FUNCTION_BLOCK FB_NanotecPD_Power
VAR_INPUT
	bExecute : BOOL;
END_VAR
VAR_OUTPUT
	bBusy 		: BOOL;
	bError 		: BOOL;
	nErrorId 	: ERRORID;	
END_VAR
VAR_IN_OUT
	pHwRef : POINTER TO FB_HwRefNanotecPD; 
END_VAR
VAR
	nState : USINT;
	fbSdoWrite : FB_SDO_WRITE;
END_VAR

//Achtung, anders als bei TMCM-Controllern wird die Statemachine des Controller hier nur bis "SwitchedOn" durchlaufen.
//"OperationEnabled" wird erst nach dem Setzen des Modes gesetzt. Jedes Ändern des Modes erfordert eine Rückkehr zu "SwitchedOn"
IF bExecute THEN
	IF nState = 0 THEN
		bBusy := TRUE;
		CASE pHwRef^.M_GetDS402State() OF
			E_CoDS402States.DS402STATE_Fault:
				pHwRef^.nControlword := 153;	//Reset Error
			E_CoDS402States.DS402STATE_SwitchOnDisabled:
				nState := 1;
			E_CoDS402States.DS402STATE_ReadyToSwitchOn:
				pHwRef^.nControlword := 0;	//Transition 7 in DS402 statemachine -> geht in Switch on disabled
				nState := 1;
			E_CoDS402States.DS402STATE_SwitchedOn:
				pHwRef^.nControlword := 0;	//Transition 10 in DS402 statemachine -> geht in Switch on disabled
				nState := 1;
			E_CoDS402States.DS402STATE_OperationEnabled:
				pHwRef^.nControlword := 0;	//Shutdown
				nState := 1;
			E_CoDS402States.DS402STATE_NotReadyToSwitchOn:
				nErrorId := E_ErrorIdDS402.ERRORID_NotReadyToSwitchOn;
				nState := 99;
		END_CASE
 	END_IF
	
	CASE nState OF
		1:	//Change ro "Ready to switched on"
			pHwRef^.nControlword := 6;
			nState := 2;
			
		2:	//State = "Ready to switched on" ? -> Switch on
			IF pHwRef^.M_GetDS402State() = E_CoDS402States.DS402STATE_ReadyToSwitchOn THEN
				pHwRef^.nControlword := 7;
				nState := 3;
			ELSIF pHwRef^.M_GetDS402State() = E_CoDS402States.DS402STATE_Fault THEN
				nErrorId := E_ErrorIdDS402.ERRORID_FaultState;
				nState := 99;
			END_IF
			
		3:	//State = "Switched on" ?
			IF pHwRef^.M_GetDS402State() = E_CoDS402States.DS402STATE_SwitchedOn THEN
				//pHwRef^.nDriveSubMode := 1;
				nState := 80;
			ELSIF pHwRef^.M_GetDS402State() = E_CoDS402States.DS402STATE_Fault THEN
				nErrorId := E_ErrorIdDS402.ERRORID_FaultState;
				nState := 99;
			END_IF
			
	END_CASE
	
	IF nState >= 80 THEN
		bBusy := FALSE;
		IF nState = 99 THEN
			bError := TRUE;
		END_IF
	END_IF
	
ELSE
	bError := FALSE;
	nErrorId := 0;
	nState := 0;
END_IF

END_FUNCTION_BLOCK

(* stored: Version 1.1.0.1, ProductVersion 3.1.4024.11
   POU FB_NanotecPD_Power: Id {e2a422db-98d6-485e-aeb9-b80444d17502}, SpecialFunc None *)
